PROGRAM A10_LAB_Duplicat
VAR
	bInit	: BOOL;
	rtInit	: R_TRIG;
	
	bExecuteInit	: BOOL;
	bExecuteDup		: BOOL;
	bExecuteUpdate	: BOOL;
	bExecuteVal		: BOOL;
	bExecuteFinal	: BOOL;
	
	nOACFilesBlocked		: UINT;
	nOCVFilesBlocked		: UINT;
	
	rtExecute	: R_TRIG;
	
	//aOuters 	: ARRAY[1..3] OF ST_LAB_OuterData;
	
	nOuterIndex			: INT;
	nPackIndex			: INT;
	nOuterCheckIndex	: INT;
	nPackCheckIndex		: INT;


	nLastOuterIndexValue		: INT;
	nLastPackIndexValue			: INT;
	
	fbInitialiseCaseData	: FB_CASE_InitialiseData;
	fbCaseDuplicatCheck		: FB_CASE_DuplicatCheck;
	fbDuplicateUpdateToDB	: FB_CASE_DuplicateUpdateToDB;
	fbValidateCaseContent	: FB_CASE_ValidateContent;
	fbFinaliseData			: FB_CASE_FinaliseData;
	
	bCACValid			: BOOL;
	bCACInvalid			: BOOL;
	sRejectCode				: T_MaxString;
	sCaseContent			: T_LongSTRING;
	bIsDuplicateOuters		: BOOL;
	bIsDuplicatePacks		: BOOL;
	bDoorOpen				: BOOL;
END_VAR
VAR CONSTANT
		
	nMAX_OUTER	: INT :=3;
	nMAX_PACK	: INT :=3;
END_VAR


rtInit(CLK:=bInit);

IF rtInit.Q THEN
	Initialisation(aOuters, aLabCACData);
END_IF

InitCaseData();

DupCheck();

aOCVDataDB_LAB.bDone 	:= TRUE;
aOACDataDB_LAB.bDone	:= TRUE;

UpdateDB();

ValidateCaseData();

FinalCaseData();

(*
rtExecute(CLK:=bExecute);

IF rtExecute.Q THEN
	
	FOR  nOuterIndex :=1 TO nMAX_OUTER DO
		//////////////////////
		FOR nOuterCheckIndex := nOuterIndex + 1 TO nMAX_OUTER DO
			
			nLastOuterIndexValue	:= nOuterCheckIndex;
			 IF aOuters[nOuterIndex].sOuterCode = aOuters[nOuterCheckIndex].sOuterCode  THEN
				 
				aOuters[nOuterIndex].nOuterRejectID			:= 200;
				aOuters[nOuterCheckIndex].nOuterRejectID	:= 200;
			 END_IF
		END_FOR
		///////////////////////////
		FOR  nPackIndex :=1 TO nMAX_PACK DO
			FOR nPackCheckIndex := nPackIndex + 1  TO nMAX_PACK DO
				
				nLastPackIndexValue	:= nPackCheckIndex;
				 IF aOuters[nOuterIndex].aPacks[nPackIndex].sPackCode = aOuters[nOuterIndex].aPacks[nPackCheckIndex].sPackCode THEN
					 
					aOuters[nOuterIndex].aPacks[nPackIndex].nPackRejectID		:= 100;
					aOuters[nOuterIndex].aPacks[nPackCheckIndex].nPackRejectID	:= 100;
				END_IF
			END_FOR
			
			FOR nOuterCheckIndex := nOuterIndex + 1 TO nMAX_OUTER DO
				FOR nPackCheckIndex := 1  TO nMAX_PACK DO
					
					IF aOuters[nOuterIndex].aPacks[nPackIndex].sPackCode = aOuters[nOuterCheckIndex].aPacks[nPackCheckIndex].sPackCode THEN
					 
						aOuters[nOuterIndex].aPacks[nPackIndex].nPackRejectID		:= 100;
						aOuters[nOuterCheckIndex].aPacks[nPackCheckIndex].nPackRejectID	:= 100;
					END_IF
				END_FOR
			END_FOR
				
		END_FOR
		///////////////////////////////
	END_FOR
END_IF	
		*)
	(*	IF stOuterStatus.stOACData.PackCodeStatus[nPackIndex].5 OR stOuterStatus.stOACData.PackCodeStatus[nPackIndex].6 THEN

			FOR nCheckIndex :=1 TO cMAX_PACKS_PER_OUTER DO

				IF stOuterStatus.stOACData.PackCode[nPackIndex] = stLastOuterStatus.stOACData.PackCode[nCheckIndex] THEN

					stOuterStatus.nStatus.22 := TRUE;
					stOuterStatus.sDataSourceTracker  := 'PK_DUPLIC';

					stLastOuterStatus.nStatus.22 := TRUE;
					stLastOuterStatus.sDataSourceTracker  := 'PK_DUPLIC';

					EXIT;
				END_IF
			END_FOR
			EXIT;
		END_IF
	END_FOR*)

ACTION DupCheck:
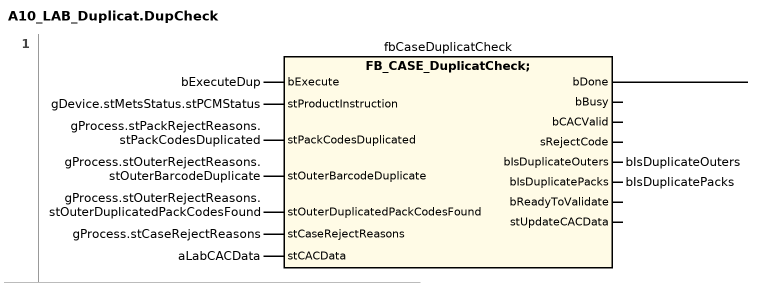
// NETWORK 1
fbCaseDuplicatCheck(
    bExecute := bExecuteDup,
    stProductInstruction := gDevice.stMetsStatus.stPCMStatus,
    stPackCodesDuplicated := gProcess.stPackRejectReasons.stPackCodesDuplicated,
    stOuterBarcodeDuplicate := gProcess.stOuterRejectReasons.stOuterBarcodeDuplicate,
    stOuterDuplicatedPackCodesFound := gProcess.stOuterRejectReasons.stOuterDuplicatedPackCodesFound,
    stCaseRejectReasons := gProcess.stCaseRejectReasons,
    stCACData := aLabCACData,
    bIsDuplicateOuters => bIsDuplicateOuters,
    bIsDuplicatePacks => bIsDuplicatePacks); // FB_CASE_DuplicatCheck;
END_ACTION

ACTION FinalCaseData:
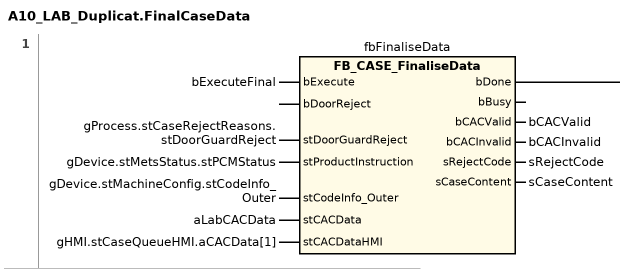
// NETWORK 1
fbFinaliseData(
    bExecute := bExecuteFinal,
    stDoorGuardReject := gProcess.stCaseRejectReasons.stDoorGuardReject,
    stProductInstruction := gDevice.stMetsStatus.stPCMStatus,
    stCodeInfo_Outer := gDevice.stMachineConfig.stCodeInfo_Outer,
    stCACData := aLabCACData,
    stCACDataHMI := gHMI.stCaseQueueHMI.aCACData[1],
    bCACValid => bCACValid,
    bCACInvalid => bCACInvalid,
    sRejectCode => sRejectCode,
    sCaseContent => sCaseContent); // FB_CASE_FinaliseData
END_ACTION

ACTION InitCaseData:
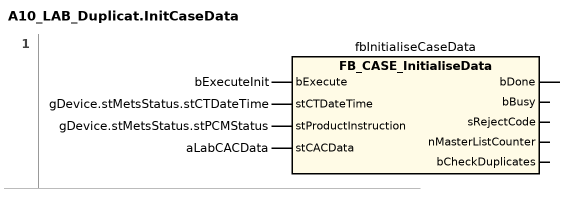
// NETWORK 1
fbInitialiseCaseData(
    bExecute := bExecuteInit,
    stCTDateTime := gDevice.stMetsStatus.stCTDateTime,
    stProductInstruction := gDevice.stMetsStatus.stPCMStatus,
    stCACData := aLabCACData); // FB_CASE_InitialiseData
END_ACTION

METHOD PRIVATE Initialisation
VAR_INPUT
END_VAR
VAR_IN_OUT
	aOuters 	: ARRAY[1..3] OF ST_LAB_OuterData;
	aLabCACData	: ST_CAC_Data;
END_VAR
VAR
	nOuterIndex			: INT;
	nPackIndex			: INT;
END_VAR
(*aOuters[1].sOuterCode	:=	'OUTER1';
aOuters[1].nOuterStatus := 5;

aOuters[1].aPacks[1].sPackCode		:= 'PACK01OUTER1';
aOuters[1].aPacks[1].nPackStatus	:= 5;
aOuters[1].aPacks[2].sPackCode		:= 'PACK02OUTER1';
aOuters[1].aPacks[2].nPackStatus	:= 5;
aOuters[1].aPacks[3].sPackCode		:= 'PACK02OUTER1';
aOuters[1].aPacks[3].nPackStatus	:= 5;

aOuters[2].sOuterCode	:= 'OUTER2';
aOuters[2].nOuterStatus := 5;

aOuters[2].aPacks[1].sPackCode		:= 'PACK01OUTER2';
aOuters[2].aPacks[1].nPackStatus	:= 5;
aOuters[2].aPacks[2].sPackCode		:= 'PACK02OUTER2';
aOuters[2].aPacks[2].nPackStatus	:= 5;
aOuters[2].aPacks[3].sPackCode		:= 'PACK02OUTER2';
aOuters[2].aPacks[3].nPackStatus	:= 5;

aOuters[3].sOuterCode	:= 'OUTER3';
aOuters[3].nOuterStatus := 5;

aOuters[3].aPacks[1].sPackCode		:= 'PACK01OUTER3';
aOuters[3].aPacks[1].nPackStatus	:= 5;
aOuters[3].aPacks[2].sPackCode		:= 'PACK02OUTER3';
aOuters[3].aPacks[2].nPackStatus	:= 5;
aOuters[3].aPacks[3].sPackCode		:= 'PACK02OUTER3';
aOuters[3].aPacks[3].nPackStatus	:= 5;
*)

MEMSET(ADR(aLabCACData), 16#00, SIZEOF(aLabCACData));

aLabCACData.NumberOfOuters			:= gDevice.stMetsStatus.stPCMStatus.nOutersPerCase;
aLabCACData.CodingAndTrackingMode	:= gDevice.stMetsStatus.stPCMStatus.nOpMode;
aLabCACData.RetailSKU				:= gDevice.stMetsStatus.stPCMStatus.sRetailSKU;

FOR nOuterIndex := 1 TO cMAX_OUTERS_PER_CASE BY 1 DO
	
	aLabCACData.Outer[nOuterIndex].Barcode 					:= CONCAT('OUTER_', INT_TO_STRING(nOuterIndex));
	aLabCACData.Outer[nOuterIndex].NumberOfPacks 			:= gDevice.stMetsStatus.stPCMStatus.nPacksPerOuter;
	aLabCACData.Outer[nOuterIndex].NumberOfLinkedPacks 		:= gDevice.stMetsStatus.stPCMStatus.nPacksPerOuter;
	aLabCACData.Outer[nOuterIndex].AcceptanceLevel 			:= gDevice.stMetsStatus.stPCMStatus.nPacksPerOuter;
	aLabCACData.Outer[nOuterIndex].CodingAndTrackingMode	:= gDevice.stMetsStatus.stPCMStatus.nOpMode;
	aLabCACData.Outer[nOuterIndex].OuterRejectCode			:= 'OK';
	
	FOR  nPackIndex :=1 TO cMAX_PACKS_PER_OUTER BY 1 DO
		aLabCACData.Outer[nOuterIndex].PackCode[nPackIndex] := F_CONCAT3(aLabCACData.Outer[nOuterIndex].Barcode,'_PACK_', INT_TO_STRING(nPackIndex));
		IF nPackIndex = 1 THEN
			aLabCACData.Outer[nOuterIndex].AggregationCodes[1]	:= aLabCACData.Outer[nOuterIndex].PackCode[nPackIndex];
		END_IF
		IF nPackIndex = 2 THEN
			aLabCACData.Outer[nOuterIndex].AggregationCodes[2]	:= aLabCACData.Outer[nOuterIndex].PackCode[nPackIndex];
		END_IF
		aLabCACData.Outer[nOuterIndex].PackCodeStatus[nPackIndex].5 := TRUE;
		aLabCACData.Outer[nOuterIndex].PackRejectCode[nPackIndex]	:= 'OK';
	END_FOR
END_FOR
END_METHOD

ACTION UpdateDB:
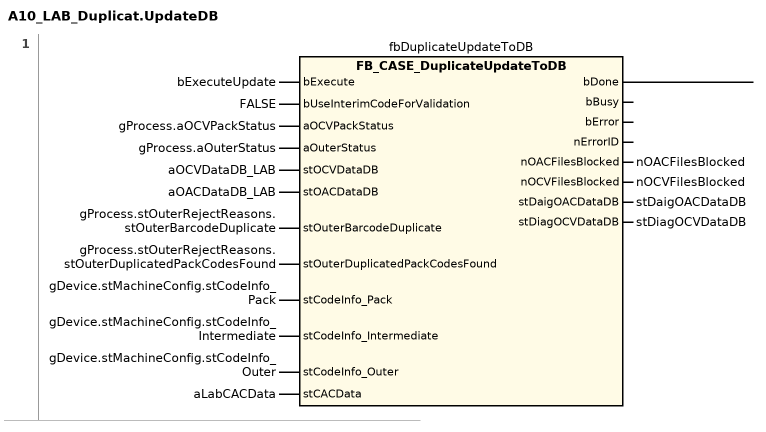
// NETWORK 1
fbDuplicateUpdateToDB(
    bExecute := bExecuteUpdate,
    bUseInterimCodeForValidation := FALSE,
    aOCVPackStatus := gProcess.aOCVPackStatus,
    aOuterStatus := gProcess.aOuterStatus,
    stOCVDataDB := aOCVDataDB_LAB,
    stOACDataDB := aOACDataDB_LAB,
    stOuterBarcodeDuplicate := gProcess.stOuterRejectReasons.stOuterBarcodeDuplicate,
    stOuterDuplicatedPackCodesFound := gProcess.stOuterRejectReasons.stOuterDuplicatedPackCodesFound,
    stCodeInfo_Pack := gDevice.stMachineConfig.stCodeInfo_Pack,
    stCodeInfo_Intermediate := gDevice.stMachineConfig.stCodeInfo_Intermediate,
    stCodeInfo_Outer := gDevice.stMachineConfig.stCodeInfo_Outer,
    stCACData := aLabCACData,
    nOACFilesBlocked => nOACFilesBlocked,
    nOCVFilesBlocked => nOCVFilesBlocked,
    stDaigOACDataDB => stDaigOACDataDB,
    stDiagOCVDataDB => stDiagOCVDataDB); // FB_CASE_DuplicateUpdateToDB
END_ACTION

ACTION ValidateCaseData:
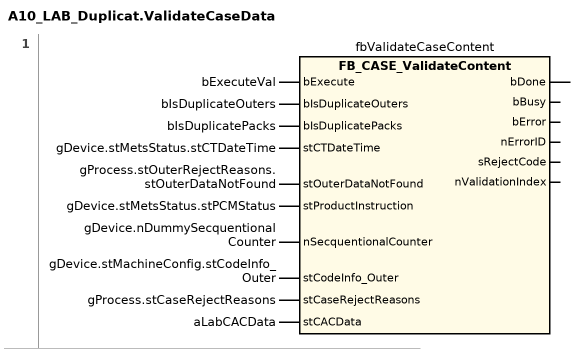
// NETWORK 1
fbValidateCaseContent(
    bExecute := bExecuteVal,
    bIsDuplicateOuters := bIsDuplicateOuters,
    bIsDuplicatePacks := bIsDuplicatePacks,
    stCTDateTime := gDevice.stMetsStatus.stCTDateTime,
    stOuterDataNotFound := gProcess.stOuterRejectReasons.stOuterDataNotFound,
    stProductInstruction := gDevice.stMetsStatus.stPCMStatus,
    nSecquentionalCounter := gDevice.nDummySecquentionalCounter,
    stCodeInfo_Outer := gDevice.stMachineConfig.stCodeInfo_Outer,
    stCaseRejectReasons := gProcess.stCaseRejectReasons,
    stCACData := aLabCACData); // FB_CASE_ValidateContent
END_ACTION

END_PROGRAM

(* stored: Version 1.1.0.1
   POU A10_LAB_Duplicat: Id {0365173a-a22a-44dc-95f2-c86f7430a9c0}, SpecialFunc None
   Action DupCheck: Id {eabea021-2b3c-4fbc-b9e9-2b8d09e09b09}
   Action FinalCaseData: Id {2d535783-b4da-45d2-a4e5-1e9edf679954}
   Action InitCaseData: Id {10890e53-dae4-43ed-ac33-b9ddb5fbef90}
   Method Initialisation: Id {671f1c5a-4441-4f61-aefb-2a5d3dc1257e}
   Action UpdateDB: Id {6121d8f3-7e88-4fe8-9f15-4bc16ea9068d}
   Action ValidateCaseData: Id {dd1ad1e3-da8c-4ab1-bbed-3544976742af} *)
